  def rq_current_pos_norm(gripper_socket="1"):
      pos_gripper = rq_current_pos(gripper_socket)
      pos_norm = gripper_to_norm(pos_gripper)
      return pos_norm
  end

  def gripper_to_norm(value_gripper):
      value_norm = (value_gripper / 255) * 100
      return floor(value_norm)
  end

  def norm_to_gripper(value_norm):
      value_gripper = (value_norm / 100) * 255
      return ceil(value_gripper)
  end

  def rq_get_position():
      return rq_current_pos_norm()
  end

  def rq_gripper_led_on(gripper_socket="1"):
      rq_set_var("LBP",0, gripper_socket)
  end

  def rq_gripper_led_off(gripper_socket="1"):
      rq_set_var("LBP",1, gripper_socket)
      rq_set_var("LRD",0, gripper_socket)
      rq_set_var("LBL",0, gripper_socket)
      rq_set_var("LGN",0, gripper_socket)
  end

  def rq_gripper_led_force_red(gripper_socket="1"):
      rq_set_var("LBP",1, gripper_socket)
      rq_set_var("LRD",1, gripper_socket)
      rq_set_var("LBL",0, gripper_socket)
      rq_set_var("LGN",0, gripper_socket)
  end

  def rq_gripper_led_force_blue(gripper_socket="1"):
      rq_set_var("LBP",1, gripper_socket)
      rq_set_var("LRD",0, gripper_socket)
      rq_set_var("LBL",1, gripper_socket)
      rq_set_var("LGN",0, gripper_socket)
  end

  def rq_gripper_led_force_green(gripper_socket="1"):
      rq_set_var("LBP",1, gripper_socket)
      rq_set_var("LRD",0, gripper_socket)
      rq_set_var("LBL",0, gripper_socket)
      rq_set_var("LGN",1, gripper_socket)
  end

  def rq_gripper_led_force_purple(gripper_socket="1"):
      rq_set_var("LBP",1, gripper_socket)
      rq_set_var("LRD",1, gripper_socket)
      rq_set_var("LBL",1, gripper_socket)
      rq_set_var("LGN",0, gripper_socket)
  end

  ############################################
  # mm/inches functions
  ############################################
  gripper_closed_norm = [100, 100, 100, 100]
  gripper_open_norm = [0, 0, 0, 0]
  gripper_closed_mm = [0, 0, 0, 0]
  gripper_open_mm = [50, 50, 50, 50]

  def rq_current_pos_mm(gripper_socket=1):
      pos_gripper = rq_current_pos(gripper_socket)
      pos_mm = gripper_to_mm(pos_gripper, gripper_socket)
      return round_value_2_dec(pos_mm)
  end

  def rq_current_pos_inches(gripper_socket=1):
      pos_gripper = rq_current_pos(gripper_socket)
      pos_mm = gripper_to_mm(pos_gripper, gripper_socket)
      pos_in = pos_mm / 25.4
      return round_value_2_dec(pos_in)
  end

  def rq_move_mm(pos_mm, gripper_socket=1):
      pos_gripper = mm_to_gripper(pos_mm, gripper_socket)
      rq_move(pos_gripper, gripper_socket)
  end

  def rq_move_and_wait_mm(pos_mm, gripper_socket=1):
      pos_gripper = mm_to_gripper(pos_mm, gripper_socket)
      rq_move_and_wait(pos_gripper, gripper_socket)
  end

  def rq_move_inches(pos_in, gripper_socket=1):
      pos_mm = pos_in * 25.4
      rq_move_mm(pos_mm, gripper_socket)
  end

  def rq_move_and_wait_inches(pos_in, gripper_socket=1):
      pos_mm = pos_in * 25.4
      rq_move_and_wait_mm(pos_mm, gripper_socket)
  end

  def get_closed_norm(gripper_socket):
      return gripper_closed_norm[gripper_socket - 1]
  end

  def get_open_norm(gripper_socket):
      return gripper_open_norm[gripper_socket - 1]
  end

  def get_closed_mm(gripper_socket):
      return gripper_closed_mm[gripper_socket - 1]
  end

  def get_open_mm(gripper_socket):
      return gripper_open_mm[gripper_socket - 1]
  end

  def set_closed_norm(closed_norm, gripper_socket):
      gripper_closed_norm[gripper_socket - 1] = closed_norm
  end

  def set_open_norm(open_norm, gripper_socket):
      gripper_open_norm[gripper_socket - 1] = open_norm
  end

  def set_closed_mm(closed_mm, gripper_socket):
      gripper_closed_mm[gripper_socket - 1] = closed_mm
  end

  def set_open_mm(open_mm, gripper_socket):
      gripper_open_mm[gripper_socket - 1] = open_mm
  end

  def gripper_to_mm(value_gripper, gripper_socket):
      closed_norm = get_closed_norm(gripper_socket)
      open_norm = get_open_norm(gripper_socket)
      closed_mm = get_closed_mm(gripper_socket)
      open_mm = get_open_mm(gripper_socket)

      value_norm = (value_gripper / 255) * 100

      slope = (closed_mm - open_mm) / (closed_norm - open_norm)
      value_mm = slope * (value_norm - closed_norm) + closed_mm

      if (value_mm > open_mm):
          value_mm_limited = open_mm
      elif (value_mm < closed_mm):
          value_mm_limited = closed_mm
      else:
          value_mm_limited = value_mm
      end

      return value_mm_limited
  end

  def mm_to_gripper(value_mm, gripper_socket):
      closed_norm = get_closed_norm(gripper_socket)
      open_norm = get_open_norm(gripper_socket)
      closed_mm = get_closed_mm(gripper_socket)
      open_mm = get_open_mm(gripper_socket)

      slope = (closed_norm - open_norm) / (closed_mm - open_mm)
      value_norm = (value_mm - closed_mm) * slope + closed_norm

      value_gripper = value_norm * 255 / 100

      if (value_gripper > 255):
          value_gripper_limited = 255
      elif (value_gripper < 0):
          value_gripper_limited = 0
      else:
          value_gripper_limited = round_value(value_gripper)
      end

      return value_gripper_limited
  end

  def round_value(value):
      value_mod = value % 1

      if(value_mod < 0.5):
          return floor(value)
      else:
          return ceil(value)
      end
  end

  def round_value_2_dec(value):
      value_x_100 = value * 100
      value_x_100_rounded = round_value(value_x_100)
      return value_x_100_rounded / 100
  end

  def clear_socket_buffer(gripper_socket="1", read_timeout = 0.1):
      rq_comm_clear_socket_buffer_enabled[rq_socket_to_index(gripper_socket)] = True
  end

  def rq_gripper_id_to_ascii(gripper_id):
      if(gripper_id == "1"):
          return 57
      elif(gripper_id == "2"):
          return 50
      elif(gripper_id == "3"):
          return 51
      elif(gripper_id == "4"):
          return 52
      end
  end

  def scale(value, rawRange, scaledRange):
      def computeSlope(inputRange, outputRange):
          outputRangeDelta = outputRange[1] - outputRange[0]
          inputRangeDelta = inputRange[1] - inputRange[0]

          if (inputRangeDelta == 0):
              return 0
          else:
              return outputRangeDelta / inputRangeDelta
          end
      end

      def computeIntercept(slope, inputRange, outputRange):
          return outputRange[0] - (slope * inputRange[0])
      end

      def clipScaledValue(outputScaledValue, outputRange):
          if (outputRange[0] < outputRange[1]):
              return clipWhenLowerLimitIsLessThanHigher(outputScaledValue, outputRange)
          else:
              return clipWhenLowerLimitIsGreaterThanHigherLimit(outputScaledValue, outputRange)
          end
      end

      def clipWhenLowerLimitIsGreaterThanHigherLimit(outputScaledValue, outputRange):
          if (outputScaledValue < outputRange[1]):
              return outputRange[1]
          elif (outputScaledValue > outputRange[0]):
              return outputRange[0]
          else:
              return outputScaledValue
          end
      end

      def clipWhenLowerLimitIsLessThanHigher(outputScaledValue, outputRange):
          if (outputScaledValue < outputRange[0]):
              return outputRange[0]
          elif (outputScaledValue > outputRange[1]):
              return outputRange[1]
          else:
              return outputScaledValue
          end
      end

      slope = computeSlope(rawRange, scaledRange)
      intercept = computeIntercept(slope, rawRange, scaledRange)
      scaledValue = slope * value + intercept
      return clipScaledValue(scaledValue, scaledRange)
  end

  def limit(value, range):
      return scale(value, range, range)
  end


  rq_init_comm_if_connected(9, "1")
  rq_init_comm_if_connected(2, "2")
  rq_init_comm_if_connected(3, "3")
  rq_init_comm_if_connected(4, "4")
  rq_print_connected_grippers()
  rq_gripper_communication_thread = run rq_gripper_communication()
  set_closed_norm(100.0, 1)
  set_open_norm(0.0, 1)
  set_closed_mm(0.0, 1)
  set_open_mm(50.0, 1)
  set_closed_norm(100.0, 2)
  set_open_norm(0.0, 2)
  set_closed_mm(0.0, 2)
  set_open_mm(50.0, 2)
  set_closed_norm(100.0, 3)
  set_open_norm(0.0, 3)
  set_closed_mm(0.0, 3)
  set_open_mm(50.0, 3)
  set_closed_norm(100.0, 4)
  set_open_norm(0.0, 4)
  set_closed_mm(0.0, 4)
  set_open_mm(50.0, 4)
  rq_current_limit_enabled = False
  while(not rq_gripper_communication_thread_started):
      sleep(0.008)
  end
  # end: URCap Installation Node
  $ 1 "BeforeStart"
  # begin: URCap Program Node
  #   Source: Robotiq_Grippers, 1.8.9.14887, Robotiq Inc.
  #   Type: Gripper Activate
  $ 2 "Gripper Reset and Activate"

  kill rq_gripper_communication_thread
  rq_gripper_communication_thread_started = False
  rq_close_gripper_socket("1")
  rq_close_gripper_socket("2")
  rq_close_gripper_socket("3")
  rq_close_gripper_socket("4")

  rq_init_comm_if_connected(9, "1")
  rq_init_comm_if_connected(2, "2")
  rq_init_comm_if_connected(3, "3")
  rq_init_comm_if_connected(4, "4")
  rq_print_connected_grippers()
  rq_gripper_communication_thread = run rq_gripper_communication()

  while(not rq_gripper_communication_thread_started):
      sleep(0.008)
  end

  rq_set_max_current_for_all_grippers()

  reset_and_activate = True

  rq_activate_all_grippers(True)
  # end: URCap Program Node
  # begin: URCap Program Node
  #   Source: Robotiq_Grippers, 1.8.9.14887, Robotiq Inc.
  #   Type: Gripper
  $ 3 "Gripper Open (1)"
  if not(gripper_connected[0]):
    popup("Gripper 1 must be connected to run this program.", "No connection", False, True, True)
  end
  if not(rq_is_gripper_activated("1")):
    popup("Gripper 1 is not activated. Go to Installation tab > Gripper to activate it and run the program again.", "Not activated", False, True, True)
  end
  rq_set_pos_spd_for(0, 255, 0, "1")
  rq_wait_pos_spe_for_request(0, 255, 0, "1")
  rq_go_to("1")
  rq_wait("1")
  # end: URCap Program Node
  $ 4 "MoveJ"
  $ 5 "Waypoint_h" "breakAfter"
  movej(get_inverse_kin(p[-.113000086719, -.297659967309, .156244786893, -.002737062845, -3.140527714900, -.001955413206], qnear=[4.712365150451953, -1.5707362333879464, -1.5708439985859712, -1.5708563963519486, 1.570766806602113, 6.283185307179586]), a=1.3962634015954636, v=1.0471975511965976)
  while (True):
    $ 6 "Robot Program"
    $ 7 "MoveJ"
    $ 8 "snap_pos" "breakAfter"
    movej(get_inverse_kin(p[-.094078273465, -.366179396653, .154237533344, .079491017081, -3.139371350249, .025270080383], qnear=[4.764800071715875, -1.8153126875508736, -1.3089636007887977, -1.5708563963525641, 1.5707963267948966, 6.283185307179586]), a=1.3962634015954636, v=1.0471975511965976)
    # begin: URCap Program Node
    #   Source: Robotiq_Wrist_Camera, 1.11.3.13312, Robotiq Inc.
    #   Type: Cam Locate
    $ 9 "Cam Locate"

    ###########################################
    #######VisionLocate node start########

    f=[0,0.0,0.0,0.0,0.0,0.0,0.0,0]
    object_location=p[0.0,0.0,0.0,0.0,0.0,0.0]
    feature_pose_to_restore_17539 = Calib_1
    if (cam_locate_monitor.isCaptureNeeded("17539")):
      movej([4.875949382781982, -1.7095311323748987, -1.2673834005938929, -1.2232511679278772, 1.4940849542617798, 6.425290499125616])
      # Offset in translation only.
      snapshot_position_offset[3] = 0
      snapshot_position_offset[4] = 0
      snapshot_position_offset[5] = 0
      T_camera_in_flange = p[0, 0, 0, 0, 0, 0] # enlever une fois que l'enseignement du modele sera fait en faisant un movetool avec la pose de la camera dans le repere de la flange. Pour l'instant, on suppose que la camera est situee directement sur la flange.
      tool_17539 = get_T_in_base_from_flange(T_camera_in_flange)
      tool_17539 = pose_sub(tool_17539, snapshot_position_offset)
      snapshot_position = p[-0.0593039, -0.372524, 0.398348, 3.82588E-4, 3.03598, -0.801907]
      textmsg("expected snapshot position : ", snapshot_position)
      diff = pose_sub(tool_17539, snapshot_position)
      textmsg("diff = ", diff)
      is_at_snapshot_position = norm([diff[0], diff[1], diff[2]]) < 0.002
      is_at_snapshot_position = is_at_snapshot_position and (norm([diff[3], diff[4], diff[5]]) < 0.005)
      textmsg("is_at_snapshot_position = ", is_at_snapshot_position)
      is_snapshot_position_offset = norm(snapshot_position_offset) != 0
      is_at_snapshot_position = is_at_snapshot_position or ignore_snapshot_position
      if not(is_at_snapshot_position):
        popup("Robot is not at Snapshot Position. Add Move instruction to Snapshot Position before Camera Locate node.. Error code: [UCC-8]", warning = False, error = True)
        halt
      end
      f_17539 = xmlrpc_server.findmodel("contextName-17539", tool_17539[0], tool_17539[1], tool_17539[2], tool_17539[3], tool_17539[4], tool_17539[5])
      cam_locate_monitor.setFindModelResult("17539", f_17539)
      canSaveImage = True
      logging_service.publish("FIND_MODEL", f_17539)
      cam_locate_monitor.setCurrentObjectIndex("17539", 0)
    end
    # begin: URCap Program Node
    #   Source: Robotiq_Wrist_Camera, 1.11.3.13312, Robotiq Inc.
    #   Type: Cam Locate Loop
    $ 10 "For next object" "noBreak"
    object_teaching_location_17539 = p[-0.02075112124421394, -0.3236393499274243, 0.03486296230814004, -0.014685885212245018, -3.1404071737658232, 0.007030576442225836]
    feature_teaching_location_17539 = p[-0.02075112124421394, -0.3236393499274243, 0.03486296230814004, -0.008776975159103011, -3.1404208322940663, 0.0070271674057956705]
    if (not cam_locate_monitor.isCaptureNeeded("17539")):
      poseAsArray = cam_locate_monitor.getCurrentObjectPoseAsArray("17539")
      current_object_location_17539 = p[poseAsArray[0], poseAsArray[1], poseAsArray[2], poseAsArray[3], poseAsArray[4], poseAsArray[5]]
      object_location = current_object_location_17539
      f[0] = cam_locate_monitor.getNumberOfObjectsFound("17539")
      f[1] = object_location[0]
      f[2] = object_location[1]
      f[3] = object_location[2]
      f[4] = object_location[3]
      f[5] = object_location[4]
      f[6] = object_location[5]
      f[7] = cam_locate_monitor.getCurrentObjectDetectionScore("17539")
      textmsg("current_object_location = ", current_object_location_17539)
      if (norm(snapshot_position_offset) != 0):
        current_object_location_17539 = pose_add(current_object_location_17539, snapshot_position_offset)
        textmsg("current_object_location after snapshot position offset = ", current_object_location_17539)
      end
      Calib_1 = pose_trans(current_object_location_17539, pose_trans(pose_inv(object_teaching_location_17539), feature_teaching_location_17539))
      $ 11 "MoveL" "noBreak"
      $ 12 "approccio_pick" "noBreak"
      movel(pose_trans(Calib_1, p[0.006323013694076283,-0.006898678056074525,-0.010891702817897003,-0.03371192314795168,0.0049811648476972906,-0.05289143713111993]), a=1.2, v=0.25)
      $ 13 "pick" "noBreak"
      movel(pose_trans(Calib_1, p[0.007675651350070442,0.0018266968921183402,0.009287617463813281,-0.03364031398551574,0.005062281550926986,-0.05295260582429572]), a=1.2, v=0.25)
      # begin: URCap Program Node
      #   Source: Robotiq_Grippers, 1.8.9.14887, Robotiq Inc.
      #   Type: Gripper
      $ 14 "Gripper Close (1)" "noBreak"
      if not(gripper_connected[0]):
        popup("Gripper 1 must be connected to run this program.", "No connection", False, True, True)
      end
      if not(rq_is_gripper_activated("1")):
        popup("Gripper 1 is not activated. Go to Installation tab > Gripper to activate it and run the program again.", "Not activated", False, True, True)
      end
      rq_set_pos_spd_for(255, 0, 0, "1")
      rq_wait_pos_spe_for_request(255, 0, 0, "1")
      rq_go_to("1")
      rq_wait("1")
      # end: URCap Program Node
      $ 15 "esci_pick" "noBreak"
      movel(pose_trans(Calib_1, p[0.006344316103646745,-0.006903435292697102,-0.010908603449111438,-0.03364528173671498,0.004950180453737306,-0.052891739388796016]), a=1.2, v=0.25)
      $ 16 "MoveJ" "noBreak"
      $ 17 "move_to_drop_rd" "noBreak"
      movej(get_inverse_kin(p[.349917549550, -.337988429001, .048126872310, -1.273202204758, 2.849627200325, -.068416807129], qnear=[5.753843307495117, -2.3336523214923304, -1.0213435331927698, -1.3090632597552698, 1.5640511512756348, 6.482863847409384]), a=1.3962634015954636, v=1.0471975511965976)
      $ 18 "MoveL" "noBreak"
      $ 19 "place" "noBreak"
      movel(p[.349896986914, -.338027887061, .031611785308, -1.273203482905, 2.849604154329, -.068491276241], a=1.2, v=0.25)
      # begin: URCap Program Node
      #   Source: Robotiq_Grippers, 1.8.9.14887, Robotiq Inc.
      #   Type: Gripper
      $ 20 "Gripper Open (1)" "noBreak"
      if not(gripper_connected[0]):
        popup("Gripper 1 must be connected to run this program.", "No connection", False, True, True)
      end
      if not(rq_is_gripper_activated("1")):
        popup("Gripper 1 is not activated. Go to Installation tab > Gripper to activate it and run the program again.", "Not activated", False, True, True)
      end
      rq_set_pos_spd_for(0, 0, 0, "1")
      rq_wait_pos_spe_for_request(0, 0, 0, "1")
      rq_go_to("1")
      rq_wait("1")
      # end: URCap Program Node
      $ 21 "Waypoint_3" "noBreak"
      movel(p[.349917549550, -.337988429001, .048126872310, -1.273202204758, 2.849627200325, -.068416807129], a=1.2, v=0.25)
      $ 22 "Waypoint_3" "noBreak"
      movej(get_inverse_kin(p[.349917549550, -.337988429001, .048126872310, -1.273202204758, 2.849627200325, -.068416807129], qnear=[5.753843307495117, -2.3336523214923304, -1.0213435331927698, -1.3090632597552698, 1.5640511512756348, 6.482863847409384]), a=1.3962634015954636, v=1.0471975511965976)
      cam_locate_monitor.incrementIndex("17539")
    end
    # end: URCap Program Node
    # begin: URCap Program Node
    #   Source: Robotiq_Wrist_Camera, 1.11.3.13312, Robotiq Inc.
    #   Type: If no object found in Camera Locate
    $ 23 "If no object found" "noBreak"
    if (not cam_locate_monitor.hasFoundObjects("17539")):
      f[0] = 0
      # begin: URCap Program Node
      #   Source: Robotiq_Wrist_Camera, 1.11.3.13312, Robotiq Inc.
      #   Type: Cam Locate
      $ 24 "Cam Locate" "noBreak"

      ###########################################
      #######VisionLocate node start########

      f=[0,0.0,0.0,0.0,0.0,0.0,0.0,0]
      object_location=p[0.0,0.0,0.0,0.0,0.0,0.0]
      feature_pose_to_restore_99554 = Calib_1
      if (cam_locate_monitor.isCaptureNeeded("99554")):
        movej([4.875949382781982, -1.7095311323748987, -1.2673834005938929, -1.2232511679278772, 1.4940849542617798, 6.425290499125616])
        # Offset in translation only.
        snapshot_position_offset[3] = 0
        snapshot_position_offset[4] = 0
        snapshot_position_offset[5] = 0
        T_camera_in_flange = p[0, 0, 0, 0, 0, 0] # enlever une fois que l'enseignement du modele sera fait en faisant un movetool avec la pose de la camera dans le repere de la flange. Pour l'instant, on suppose que la camera est situee directement sur la flange.
        tool_99554 = get_T_in_base_from_flange(T_camera_in_flange)
        tool_99554 = pose_sub(tool_99554, snapshot_position_offset)
        snapshot_position = p[-0.0593039, -0.372524, 0.398348, 3.82588E-4, 3.03598, -0.801907]
        textmsg("expected snapshot position : ", snapshot_position)
        diff = pose_sub(tool_99554, snapshot_position)
        textmsg("diff = ", diff)
        is_at_snapshot_position = norm([diff[0], diff[1], diff[2]]) < 0.002
        is_at_snapshot_position = is_at_snapshot_position and (norm([diff[3], diff[4], diff[5]]) < 0.005)
        textmsg("is_at_snapshot_position = ", is_at_snapshot_position)
        is_snapshot_position_offset = norm(snapshot_position_offset) != 0
        is_at_snapshot_position = is_at_snapshot_position or ignore_snapshot_position
        if not(is_at_snapshot_position):
          popup("Robot is not at Snapshot Position. Add Move instruction to Snapshot Position before Camera Locate node.. Error code: [UCC-8]", warning = False, error = True)
          halt
        end
        f_99554 = xmlrpc_server.findmodel("contextName-99554", tool_99554[0], tool_99554[1], tool_99554[2], tool_99554[3], tool_99554[4], tool_99554[5])
        cam_locate_monitor.setFindModelResult("99554", f_99554)
        canSaveImage = True
        logging_service.publish("FIND_MODEL", f_99554)
        cam_locate_monitor.setCurrentObjectIndex("99554", 0)
      end
      # begin: URCap Program Node
      #   Source: Robotiq_Wrist_Camera, 1.11.3.13312, Robotiq Inc.
      #   Type: Cam Locate Loop
      $ 25 "For next object" "noBreak"
      object_teaching_location_99554 = p[-0.033085168848221026, -0.3612924725286147, 0.03280792910177617, -0.014685885212238136, -3.1404071737658237, 0.007030576442314657]
      feature_teaching_location_99554 = p[-0.033085168848221026, -0.3612924725286147, 0.03280792910177617, 3.115539880768529, 0.3687589065266703, -0.002638110127252574]
      if (not cam_locate_monitor.isCaptureNeeded("99554")):
        poseAsArray = cam_locate_monitor.getCurrentObjectPoseAsArray("99554")
        current_object_location_99554 = p[poseAsArray[0], poseAsArray[1], poseAsArray[2], poseAsArray[3], poseAsArray[4], poseAsArray[5]]
        object_location = current_object_location_99554
        f[0] = cam_locate_monitor.getNumberOfObjectsFound("99554")
        f[1] = object_location[0]
        f[2] = object_location[1]
        f[3] = object_location[2]
        f[4] = object_location[3]
        f[5] = object_location[4]
        f[6] = object_location[5]
        f[7] = cam_locate_monitor.getCurrentObjectDetectionScore("99554")
        textmsg("current_object_location = ", current_object_location_99554)
        if (norm(snapshot_position_offset) != 0):
          current_object_location_99554 = pose_add(current_object_location_99554, snapshot_position_offset)
          textmsg("current_object_location after snapshot position offset = ", current_object_location_99554)
        end
        Calib_1 = pose_trans(current_object_location_99554, pose_trans(pose_inv(object_teaching_location_99554), feature_teaching_location_99554))
        $ 26 "MoveL" "noBreak"
        $ 27 "approccio_pic_1" "noBreak"
        movel(pose_trans(Calib_1, p[0.006323013694076283,-0.006898678056074525,-0.010891702817897003,-0.03371192314795168,0.0049811648476972906,-0.05289143713111993]), a=1.2, v=0.25)
        $ 28 "pick_1" "noBreak"
        movel(pose_trans(Calib_1, p[0.007675651350070442,0.0018266968921183402,0.009287617463813281,-0.03364031398551574,0.005062281550926986,-0.05295260582429572]), a=1.2, v=0.25)
        # begin: URCap Program Node
        #   Source: Robotiq_Grippers, 1.8.9.14887, Robotiq Inc.
        #   Type: Gripper
        $ 29 "Gripper Close (1)" "noBreak"
        if not(gripper_connected[0]):
          popup("Gripper 1 must be connected to run this program.", "No connection", False, True, True)
        end
        if not(rq_is_gripper_activated("1")):
          popup("Gripper 1 is not activated. Go to Installation tab > Gripper to activate it and run the program again.", "Not activated", False, True, True)
        end
        rq_set_pos_spd_for(255, 0, 0, "1")
        rq_wait_pos_spe_for_request(255, 0, 0, "1")
        rq_go_to("1")
        rq_wait("1")
        # end: URCap Program Node
        $ 30 "esci_pick_1" "noBreak"
        movel(pose_trans(Calib_1, p[0.006344316103646745,-0.006903435292697102,-0.010908603449111438,-0.03364528173671498,0.004950180453737306,-0.052891739388796016]), a=1.2, v=0.25)
        $ 31 "MoveJ" "noBreak"
        $ 32 "move_to_drop_ar" "noBreak"
        movej(get_inverse_kin(p[-.185405864287, -.449149220204, .086768730593, -.551068756796, -3.083888209426, .071071901776], qnear=[4.559679985046387, -2.307472054158346, -0.8840916792498987, -1.4744566122638147, 1.5642552375793457, 6.482540268694059]), a=1.3962634015954636, v=1.0471975511965976)
        $ 33 "MoveL" "noBreak"
        $ 34 "Waypoint_4" "noBreak"
        movel(p[-.215738295612, -.436481070915, .026939309217, -.654969051077, -3.061353739048, .075952844752], a=1.2, v=0.25)
        # begin: URCap Program Node
        #   Source: Robotiq_Grippers, 1.8.9.14887, Robotiq Inc.
        #   Type: Gripper
        $ 35 "Gripper Open (1)" "noBreak"
        if not(gripper_connected[0]):
          popup("Gripper 1 must be connected to run this program.", "No connection", False, True, True)
        end
        if not(rq_is_gripper_activated("1")):
          popup("Gripper 1 is not activated. Go to Installation tab > Gripper to activate it and run the program again.", "Not activated", False, True, True)
        end
        rq_set_pos_spd_for(0, 255, 255, "1")
        rq_wait_pos_spe_for_request(0, 255, 255, "1")
        rq_go_to("1")
        rq_wait("1")
        # end: URCap Program Node
        $ 36 "move_to_drop_ar" "noBreak"
        movel(p[-.185405864287, -.449149220204, .086768730593, -.551068756796, -3.083888209426, .071071901776], a=1.2, v=0.25)
        cam_locate_monitor.incrementIndex("99554")
      end
      # end: URCap Program Node
      # begin: URCap Program Node
      #   Source: Robotiq_Wrist_Camera, 1.11.3.13312, Robotiq Inc.
      #   Type: If no object found in Camera Locate
      $ 37 "If no object found" "noBreak"
      if (not cam_locate_monitor.hasFoundObjects("99554")):
        f[0] = 0
        $ 38 "Popup: Metti il nuovo cubo" "noBreak"
        popup("Metti il nuovo cubo", "Warning", True, False, blocking=True)
      end
      # end: URCap Program Node
      # Restore feature pose
      Calib_1 = feature_pose_to_restore_99554

      #######VisionLocate node end########
      ###########################################

      # end: URCap Program Node
    end
    # end: URCap Program Node
    # Restore feature pose
    Calib_1 = feature_pose_to_restore_17539

    #######VisionLocate node end########
    ###########################################

    # end: URCap Program Node
  end
end
